RoboDK station: 1817972 amirah husna manual.rdk

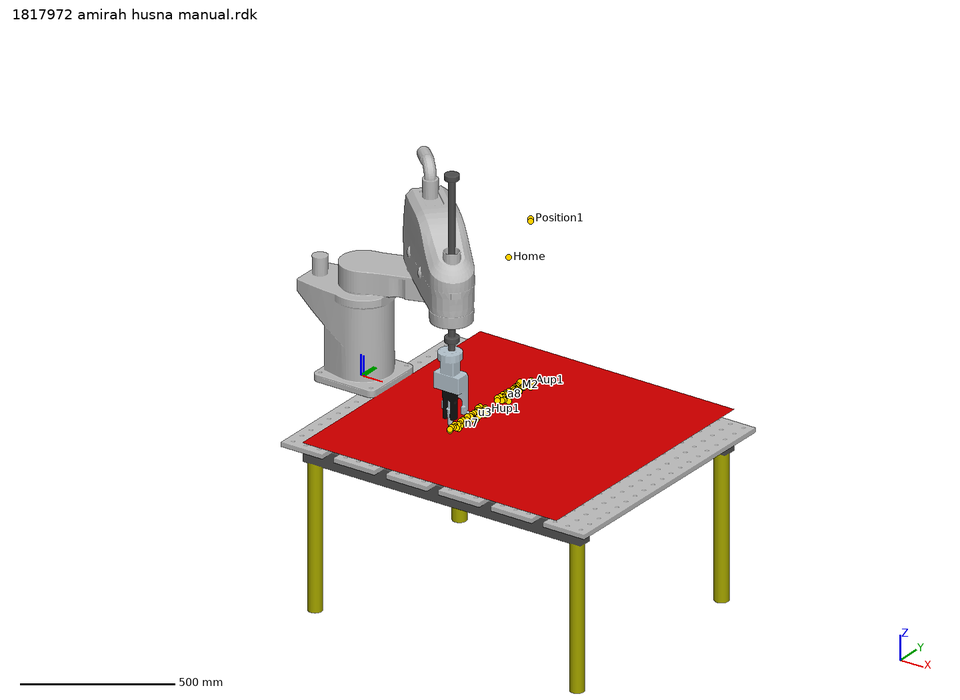
[picture v0: the station drawn from its stored meshes, robots at their saved joint values, targets as dots, program paths as lines]
Station amirah husna manual (saved by RoboDK 5.3.4). Poses are relative to the parent item; angles as X-Y-Z fixed-axis rotations.
  - frame Mitsubishi RH-12SH5535 Base at (0, 0, 0) mm
    - robot Mitsubishi RH-12SH5535: 4 axes, payload 12 kg, reach 600 mm, repeatability 0.03 mm, weight 43 kg
        modified DH rows (alpha deg, a mm, theta deg, d mm): 0, 0, 0, 0; 0, 225, 0, 0; 0, 325, 0, 0 linear; 180, 0, 0, 0
        joint limits [-140, -145, -10, -360] to [140, 145, 340, 360]; home [0, 0, 340, 0]; saved at [18.314, -60.92, 280.095, 42.606]
      - tool Gripper with pencil, TCP at (0, -10, -280) mm, rotated rx 180 ry 0 rz 0 deg, size 100 x 89.2 x 281.5 mm
  - frame Frame 2 at (-10, 0, 0) mm
    - object Object Table at (620, 0, -40) mm, size 1193.8 x 965.2 x 609.6 mm, geometry from Object Table.wrl
    - object Plane at (630, 0, 2) mm, size 1000 x 1000 x 0.5 mm, geometry from plane.sld
    - target Home (Cartesian target) at (557.97, 35.03, 564.41) mm; joints [7.617, -6.699, 291.409, -0.918] of Mitsubishi RH-12SH5535
    - target Aup1 (Cartesian target) at (473.2, 285.09, -0.83) mm, rotated rx 180 ry 0 rz 0 deg; joints [36.19, -6.243, 279.167, -29.946] of Mitsubishi RH-12SH5535
    - target A4 (Cartesian target) at (473.25, 285.09, -5.59) mm, rotated rx 180 ry 0 rz 0 deg; joints [36.081, -6.065, 274.409, -30.016] of Mitsubishi RH-12SH5535
    - target A5 (Cartesian target) at (473.25, 245.06, -5.59) mm, rotated rx 180 ry 0 rz 0 deg; joints [48.093, -32.454, 274.409, -15.638] of Mitsubishi RH-12SH5535
    - target Aup2 (Cartesian target) at (473.14, 245.06, 1.51) mm, rotated rx 180 ry 0 rz 0 deg; joints [48.146, -32.534, 281.511, -15.613] of Mitsubishi RH-12SH5535
    - target Position1 (Cartesian target) at (451.34, 310.3, 564.41) mm; joints [40.788, -10.621, 281.409, -30.167] of Mitsubishi RH-12SH5535
    - target Down1 (Cartesian target) at (451.34, 310.3, 554.41) mm; joints [48.613, -22.805, 281.409, -25.808] of Mitsubishi RH-12SH5535
    - target A1 (Cartesian target) at (493.02, 251.45, -5.59) mm, rotated rx 180 ry 0 rz 0 deg; joints [32.04, -6.116, 274.409, -25.924] of Mitsubishi RH-12SH5535
    - target A2 (Cartesian target) at (451.34, 251.57, -5.59) mm, rotated rx 180 ry 0 rz 0 deg; joints [56.255, -43.006, 274.409, -13.248] of Mitsubishi RH-12SH5535
    - target A3 (Cartesian target) at (456.2, 244.79, -5.59) mm, rotated rx 180 ry 0 rz 0 deg; joints [55.046, -42.54, 274.409, -12.506] of Mitsubishi RH-12SH5535
    - target Aup3 (Cartesian target) at (456.71, 244.79, 6.07) mm, rotated rx 180 ry 0 rz 0 deg; joints [54.857, -42.274, 286.074, -12.583] of Mitsubishi RH-12SH5535
    - target Mup1 (Cartesian target) at (476.08, 240.53, 3.16) mm, rotated rx 180 ry 0 rz 0 deg; joints [47.367, -32.207, 283.156, -15.16] of Mitsubishi RH-12SH5535
    - target M1 (Cartesian target) at (474.44, 240.53, -5.59) mm, rotated rx 180 ry 0 rz 0 deg; joints [48.113, -33.312, 274.409, -14.801] of Mitsubishi RH-12SH5535
    - target M2 (Cartesian target) at (451.34, 237.47, -5.59) mm, rotated rx 180 ry 0 rz 0 deg; joints [57.291, -46.985, 274.409, -10.306] of Mitsubishi RH-12SH5535
    - target M3 (Cartesian target) at (474.44, 230.54, -5.59) mm, rotated rx 180 ry 0 rz 0 deg; joints [49.16, -36.663, 274.409, -12.496] of Mitsubishi RH-12SH5535
    - target M4 (Cartesian target) at (451.34, 230.52, -5.59) mm, rotated rx 180 ry 0 rz 0 deg; joints [57.69, -48.777, 274.409, -8.913] of Mitsubishi RH-12SH5535
    - target M5 (Cartesian target) at (474.44, 219.74, -5.59) mm, rotated rx 180 ry 0 rz 0 deg; joints [50.032, -39.877, 274.409, -10.155] of Mitsubishi RH-12SH5535
    - target M6 (Cartesian target) at (451.34, 219.84, -5.59) mm, rotated rx 180 ry 0 rz 0 deg; joints [58.175, -51.343, 274.409, -6.833] of Mitsubishi RH-12SH5535
    - target M7 (Cartesian target) at (461.93, 215.03, -5.59) mm, rotated rx 180 ry 0 rz 0 deg; joints [54.851, -47.594, 274.409, -7.257] of Mitsubishi RH-12SH5535
    - target I1 (Cartesian target) at (472.85, 204.97, -5.59) mm, rotated rx 180 ry 0 rz 0 deg; joints [51.459, -44.57, 274.41, -6.889] of Mitsubishi RH-12SH5535
    - target I2 (Cartesian target) at (464.34, 211.06, -5.59) mm, rotated rx 180 ry 0 rz 0 deg; joints [54.191, -47.371, 274.41, -6.82] of Mitsubishi RH-12SH5535
    - target I3 (Cartesian target) at (451.34, 211.86, -5.59) mm, rotated rx 180 ry 0 rz 0 deg; joints [58.448, -53.129, 274.409, -5.318] of Mitsubishi RH-12SH5535
    - target I4 (Cartesian target) at (461.93, 203.58, -5.59) mm, rotated rx 180 ry 0 rz 0 deg; joints [55.266, -50.203, 274.409, -5.063] of Mitsubishi RH-12SH5535
    - target R1 (Cartesian target) at (470.19, 197.42, -5.59) mm, rotated rx 180 ry 0 rz 0 deg; joints [52.669, -47.637, 274.409, -5.033] of Mitsubishi RH-12SH5535
    - target R2 (Cartesian target) at (477.11, 195.12, -5.59) mm, rotated rx 180 ry 0 rz 0 deg; joints [50.312, -44.666, 274.409, -5.646] of Mitsubishi RH-12SH5535
    - target R3 (Cartesian target) at (469.73, 199.31, -5.59) mm, rotated rx 180 ry 0 rz 0 deg; joints [52.767, -47.441, 274.409, -5.326] of Mitsubishi RH-12SH5535
    - target R3.5 (Cartesian target) at (469.73, 201.5, -5.59) mm, rotated rx 180 ry 0 rz 0 deg; joints [52.694, -46.948, 274.409, -5.746] of Mitsubishi RH-12SH5535
    - target R3.55 (Cartesian target) at (471.65, 195.27, -5.59) mm, rotated rx 180 ry 0 rz 0 deg; joints [52.233, -47.396, 274.409, -4.836] of Mitsubishi RH-12SH5535
    - target R3.6 (Cartesian target) at (471.65, 190.99, -5.59) mm, rotated rx 180 ry 0 rz 0 deg; joints [52.346, -48.315, 274.409, -4.032] of Mitsubishi RH-12SH5535
    - target R4 (Cartesian target) at (474.41, 185.39, -5.59) mm, rotated rx 180 ry 0 rz 0 deg; joints [51.527, -48.134, 274.409, -3.393] of Mitsubishi RH-12SH5535
    - target R5 (Cartesian target) at (461.56, 188.8, -5.59) mm, rotated rx 180 ry 0 rz 0 deg; joints [55.692, -53.409, 274.409, -2.283] of Mitsubishi RH-12SH5535
    - target R6 (Cartesian target) at (451.34, 186.17, -5.59) mm, rotated rx 180 ry 0 rz 0 deg; joints [58.859, -58.225, 274.409, -0.634] of Mitsubishi RH-12SH5535
    - target R7 (Cartesian target) at (461.93, 176.77, -5.59) mm, rotated rx 180 ry 0 rz 0 deg; joints [55.657, -55.483, 274.409, -0.174] of Mitsubishi RH-12SH5535
    - target a1 (Cartesian target) at (471.07, 162.8, -5.59) mm, rotated rx 180 ry 0 rz 0 deg; joints [52.77, -53.89, 274.409, 1.12] of Mitsubishi RH-12SH5535
    - target a2 (Cartesian target) at (476.85, 158.23, -5.59) mm, rotated rx 180 ry 0 rz 0 deg; joints [50.897, -52.02, 274.409, 1.123] of Mitsubishi RH-12SH5535
    - target a3 (Cartesian target) at (459.52, 173.46, -5.59) mm, rotated rx 180 ry 0 rz 0 deg; joints [56.39, -57.081, 274.409, 0.692] of Mitsubishi RH-12SH5535
    - target a4 (Cartesian target) at (451.34, 169.13, -5.59) mm, rotated rx 180 ry 0 rz 0 deg; joints [58.784, -61.128, 274.409, 2.345] of Mitsubishi RH-12SH5535
    - target a5 (Cartesian target) at (460.8, 160.64, -5.59) mm, rotated rx 180 ry 0 rz 0 deg; joints [55.888, -58.649, 274.409, 2.76] of Mitsubishi RH-12SH5535
    - target a6 (Cartesian target) at (470.78, 157.7, -5.59) mm, rotated rx 180 ry 0 rz 0 deg; joints [52.816, -54.853, 274.409, 2.037] of Mitsubishi RH-12SH5535
    - target a7 (Cartesian target) at (457.33, 158.29, -5.59) mm, rotated rx 180 ry 0 rz 0 deg; joints [56.875, -60.428, 274.409, 3.553] of Mitsubishi RH-12SH5535
    - target a8 (Cartesian target) at (451.34, 154.04, -5.59) mm, rotated rx 180 ry 0 rz 0 deg; joints [58.509, -63.419, 274.409, 4.91] of Mitsubishi RH-12SH5535
    - target a9 (Cartesian target) at (461.93, 142.7, -5.59) mm, rotated rx 180 ry 0 rz 0 deg; joints [55.169, -60.819, 274.409, 5.65] of Mitsubishi RH-12SH5535
    - target h1 (Cartesian target) at (493.02, 127.33, -5.59) mm, rotated rx 180 ry 0 rz 0 deg; joints [45.116, -49.014, 274.409, 3.898] of Mitsubishi RH-12SH5535
    - target h2 (Cartesian target) at (461.93, 139.05, -5.59) mm, rotated rx 180 ry 0 rz 0 deg; joints [55.059, -61.311, 274.409, 6.252] of Mitsubishi RH-12SH5535
    - target h3 (Cartesian target) at (451.34, 136.81, -5.59) mm, rotated rx 180 ry 0 rz 0 deg; joints [57.972, -65.744, 274.409, 7.771] of Mitsubishi RH-12SH5535
    - target h4 (Cartesian target) at (477.38, 125.53, -5.59) mm, rotated rx 180 ry 0 rz 0 deg; joints [50.045, -56.573, 274.409, 6.528] of Mitsubishi RH-12SH5535
    - target h5 (Cartesian target) at (473.98, 118.78, -5.59) mm, rotated rx 180 ry 0 rz 0 deg; joints [50.804, -58.868, 274.409, 8.065] of Mitsubishi RH-12SH5535
    - target h6 (Cartesian target) at (451.34, 123.67, -5.59) mm, rotated rx 180 ry 0 rz 0 deg; joints [57.412, -67.317, 274.409, 9.905] of Mitsubishi RH-12SH5535
    - target h7 (Cartesian target) at (461.93, 108.73, -5.59) mm, rotated rx 180 ry 0 rz 0 deg; joints [53.751, -64.879, 274.409, 11.128] of Mitsubishi RH-12SH5535
    - target Updot1 (Cartesian target) at (483.42, 201.03, -1.25) mm, rotated rx 180 ry 0 rz 0 deg; joints [47.671, -39.768, 278.753, -7.903] of Mitsubishi RH-12SH5535
    - target Dot1 (Cartesian target) at (483.71, 201.03, -5.59) mm, rotated rx 180 ry 0 rz 0 deg; joints [47.559, -39.602, 274.41, -7.956] of Mitsubishi RH-12SH5535
    - target Dot2 (Cartesian target) at (482.8, 201.03, -5.59) mm, rotated rx 180 ry 0 rz 0 deg; joints [47.916, -40.127, 274.41, -7.788] of Mitsubishi RH-12SH5535
    - target Updot2 (Cartesian target) at (482.51, 201.03, -2.21) mm, rotated rx 180 ry 0 rz 0 deg; joints [48.028, -40.293, 277.786, -7.736] of Mitsubishi RH-12SH5535
    - target Hup1 (Cartesian target) at (476.08, 28.37, 0.73) mm, rotated rx 180 ry 0 rz 0 deg; joints [43.638, -64.719, 280.727, 21.082] of Mitsubishi RH-12SH5535
    - target H1 (Cartesian target) at (476.67, 28.37, -5.59) mm, rotated rx 180 ry 0 rz 0 deg; joints [43.484, -64.482, 274.409, 20.999] of Mitsubishi RH-12SH5535
    - target H2 (Cartesian target) at (481.32, 33.14, -5.59) mm, rotated rx 180 ry 0 rz 0 deg; joints [42.714, -62.4, 274.409, 19.686] of Mitsubishi RH-12SH5535
    - target H3 (Cartesian target) at (493.02, 15.59, -5.59) mm, rotated rx 180 ry 0 rz 0 deg; joints [37.726, -57.9, 274.409, 20.174] of Mitsubishi RH-12SH5535
    - target H4 (Cartesian target) at (486.33, 12.57, -5.59) mm, rotated rx 180 ry 0 rz 0 deg; joints [39.258, -60.89, 274.409, 21.632] of Mitsubishi RH-12SH5535
    - target H5 (Cartesian target) at (451.34, 26.46, -5.59) mm, rotated rx 180 ry 0 rz 0 deg; joints [49.642, -74.184, 274.409, 24.542] of Mitsubishi RH-12SH5535
    - target Hup2 (Cartesian target) at (451.16, 26.46, 2.44) mm, rotated rx 180 ry 0 rz 0 deg; joints [49.686, -74.25, 282.435, 24.564] of Mitsubishi RH-12SH5535
    - target Hup3 (Cartesian target) at (452.87, 11.87, 5.16) mm, rotated rx 180 ry 0 rz 0 deg; joints [47.616, -73.981, 285.163, 26.365] of Mitsubishi RH-12SH5535
    - target H6 (Cartesian target) at (451.34, 11.87, -5.59) mm, rotated rx 180 ry 0 rz 0 deg; joints [47.978, -74.531, 274.409, 26.553] of Mitsubishi RH-12SH5535
    - target H7 (Cartesian target) at (454.28, 14.58, -5.59) mm, rotated rx 180 ry 0 rz 0 deg; joints [47.595, -73.417, 274.409, 25.821] of Mitsubishi RH-12SH5535
    - target H8 (Cartesian target) at (490.19, 1.69, -5.59) mm, rotated rx 180 ry 0 rz 0 deg; joints [37.009, -59.39, 274.409, 22.381] of Mitsubishi RH-12SH5535
    - target Hup4 (Cartesian target) at (489.79, 1.69, -0.69) mm, rotated rx 180 ry 0 rz 0 deg; joints [37.119, -59.566, 279.311, 22.447] of Mitsubishi RH-12SH5535
    - target Hup5 (Cartesian target) at (466.33, 33.1, 0.85) mm, rotated rx 180 ry 0 rz 0 deg; joints [46.638, -68.398, 280.846, 21.76] of Mitsubishi RH-12SH5535
    - target H9 (Cartesian target) at (466.14, 33.1, -5.59) mm, rotated rx 180 ry 0 rz 0 deg; joints [46.687, -68.472, 274.409, 21.785] of Mitsubishi RH-12SH5535
    - target H10 (Cartesian target) at (469.45, 20.76, -5.59) mm, rotated rx 180 ry 0 rz 0 deg; joints [44.555, -67.576, 274.409, 23.022] of Mitsubishi RH-12SH5535
    - target H11 (Cartesian target) at (472.39, 2.61, -5.59) mm, rotated rx 180 ry 0 rz 0 deg; joints [41.773, -66.759, 274.409, 24.986] of Mitsubishi RH-12SH5535
    - target Hup6 (Cartesian target) at (471.59, 2.61, 2.6) mm, rotated rx 180 ry 0 rz 0 deg; joints [41.974, -67.074, 282.598, 25.1] of Mitsubishi RH-12SH5535
    - target uup1 (Cartesian target) at (476.74, -11.13, -1.91) mm, rotated rx 180 ry 0 rz 0 deg; joints [39.026, -65.092, 278.086, 26.065] of Mitsubishi RH-12SH5535
    - target u1 (Cartesian target) at (477.08, -11.13, -5.59) mm, rotated rx 180 ry 0 rz 0 deg; joints [38.939, -64.952, 274.409, 26.013] of Mitsubishi RH-12SH5535
    - target u2 (Cartesian target) at (459.41, -2.79, -5.59) mm, rotated rx 180 ry 0 rz 0 deg; joints [44.294, -71.763, 274.409, 27.469] of Mitsubishi RH-12SH5535
    - target u2.5 (Cartesian target) at (454.9, -4.46, -5.59) mm, rotated rx 180 ry 0 rz 0 deg; joints [45.15, -73.428, 274.409, 28.278] of Mitsubishi RH-12SH5535
    - target u3 (Cartesian target) at (451.34, -11.79, -5.59) mm, rotated rx 180 ry 0 rz 0 deg; joints [45.033, -74.724, 274.409, 29.691] of Mitsubishi RH-12SH5535
    - target u4 (Cartesian target) at (480.93, -23.56, -5.59) mm, rotated rx 180 ry 0 rz 0 deg; joints [36.395, -63.3, 274.409, 26.905] of Mitsubishi RH-12SH5535
    - target u5 (Cartesian target) at (451.34, -24.07, -5.59) mm, rotated rx 180 ry 0 rz 0 deg; joints [43.388, -74.644, 274.409, 31.257] of Mitsubishi RH-12SH5535
    - target u6 (Cartesian target) at (461.93, -36.56, -5.59) mm, rotated rx 180 ry 0 rz 0 deg; joints [39.242, -70.551, 274.409, 31.309] of Mitsubishi RH-12SH5535
    - target s1 (Cartesian target) at (480.93, -50.57, -5.59) mm, rotated rx 180 ry 0 rz 0 deg; joints [32.72, -62.657, 274.409, 29.937] of Mitsubishi RH-12SH5535
    - target s2 (Cartesian target) at (485.98, -46.68, -5.59) mm, rotated rx 180 ry 0 rz 0 deg; joints [31.998, -60.666, 274.409, 28.667] of Mitsubishi RH-12SH5535
    - target s3 (Cartesian target) at (474.44, -57.02, -5.59) mm, rotated rx 180 ry 0 rz 0 deg; joints [33.364, -65.062, 274.409, 31.697] of Mitsubishi RH-12SH5535
    - target s4 (Cartesian target) at (464.69, -51.2, -5.59) mm, rotated rx 180 ry 0 rz 0 deg; joints [36.504, -69.093, 274.409, 32.588] of Mitsubishi RH-12SH5535
    - target s4.5 (Cartesian target) at (454.51, -44.67, -5.59) mm, rotated rx 180 ry 0 rz 0 deg; joints [39.76, -73.091, 274.409, 33.331] of Mitsubishi RH-12SH5535
    - target s5 (Cartesian target) at (459.29, -36.56, -5.59) mm, rotated rx 180 ry 0 rz 0 deg; joints [39.848, -71.537, 274.409, 31.689] of Mitsubishi RH-12SH5535
    - target s6 (Cartesian target) at (451.34, -44.19, -5.59) mm, rotated rx 180 ry 0 rz 0 deg; joints [40.531, -74.25, 274.409, 33.719] of Mitsubishi RH-12SH5535
    - target s7 (Cartesian target) at (461.93, -65.82, -5.59) mm, rotated rx 180 ry 0 rz 0 deg; joints [34.927, -69.546, 274.409, 34.619] of Mitsubishi RH-12SH5535
    - target n1 (Cartesian target) at (474.05, -70.79, -5.59) mm, rotated rx 180 ry 0 rz 0 deg; joints [31.378, -64.575, 274.409, 33.197] of Mitsubishi RH-12SH5535
    - target n2 (Cartesian target) at (461.93, -65.82, -5.59) mm, rotated rx 180 ry 0 rz 0 deg; joints [34.927, -69.546, 274.409, 34.619] of Mitsubishi RH-12SH5535
    - target n3 (Cartesian target) at (451.34, -69.75, -5.59) mm, rotated rx 180 ry 0 rz 0 deg; joints [36.624, -73.27, 274.409, 36.646] of Mitsubishi RH-12SH5535
    - target n4 (Cartesian target) at (481.43, -87.32, -5.59) mm, rotated rx 180 ry 0 rz 0 deg; joints [27.001, -60.521, 274.409, 33.52] of Mitsubishi RH-12SH5535
    - target n5 (Cartesian target) at (477.62, -90.15, -5.59) mm, rotated rx 180 ry 0 rz 0 deg; joints [27.459, -61.919, 274.409, 34.46] of Mitsubishi RH-12SH5535
    - target n6 (Cartesian target) at (451.34, -83.97, -5.59) mm, rotated rx 180 ry 0 rz 0 deg; joints [34.323, -72.491, 274.409, 38.167] of Mitsubishi RH-12SH5535
    - target n7 (Cartesian target) at (461.93, -101.4, -5.59) mm, rotated rx 180 ry 0 rz 0 deg; joints [29.143, -67.34, 274.409, 38.197] of Mitsubishi RH-12SH5535
    - target aa1 (Cartesian target) at (471.07, -112.44, -5.59) mm, rotated rx 180 ry 0 rz 0 deg; joints [25.214, -62.811, 274.409, 37.597] of Mitsubishi RH-12SH5535
    - target aa2 (Cartesian target) at (476.85, -128.9, -5.59) mm, rotated rx 180 ry 0 rz 0 deg; joints [20.94, -58.766, 274.409, 37.826] of Mitsubishi RH-12SH5535
    - target aa3 (Cartesian target) at (459.52, -107.96, -5.59) mm, rotated rx 180 ry 0 rz 0 deg; joints [28.531, -67.733, 274.409, 39.203] of Mitsubishi RH-12SH5535
    - target aa4 (Cartesian target) at (451.34, -115.42, -5.59) mm, rotated rx 180 ry 0 rz 0 deg; joints [28.92, -70.157, 274.409, 41.237] of Mitsubishi RH-12SH5535
    - target aa5 (Cartesian target) at (460.8, -126.49, -5.59) mm, rotated rx 180 ry 0 rz 0 deg; joints [24.96, -65.545, 274.409, 40.585] of Mitsubishi RH-12SH5535
    - target aa6 (Cartesian target) at (470.78, -131.24, -5.59) mm, rotated rx 180 ry 0 rz 0 deg; joints [21.911, -61.062, 274.409, 39.151] of Mitsubishi RH-12SH5535
    - target aa7 (Cartesian target) at (457.33, -133.6, -5.59) mm, rotated rx 180 ry 0 rz 0 deg; joints [24.383, -66.151, 274.409, 41.768] of Mitsubishi RH-12SH5535
    - target aa8 (Cartesian target) at (451.34, -135.54, -5.59) mm, rotated rx 180 ry 0 rz 0 deg; joints [25.245, -68.209, 274.409, 42.964] of Mitsubishi RH-12SH5535
    - target aa9 (Cartesian target) at (461.93, -159.31, -5.59) mm, rotated rx 180 ry 0 rz 0 deg; joints [18.503, -61.277, 274.409, 42.774] of Mitsubishi RH-12SH5535
    - target aaup1 (Cartesian target) at (462.81, -159.31, 0.09) mm, rotated rx 180 ry 0 rz 0 deg; joints [18.314, -60.92, 280.095, 42.606] of Mitsubishi RH-12SH5535
  - Python program Code (listed below)
  - Python program WeldOn (listed below)
  - Python program WeldOff (listed below)

--- Python program Code ---
# Type help("robolink") or help("robodk") for more information
# Press F5 to run the script
# Documentation: https://robodk.com/doc/en/RoboDK-API.html
# Reference:     https://robodk.com/doc/en/PythonAPI/index.html
# Note: It is not required to keep a copy of this file, your python script is saved with the station
from robolink import *    # RoboDK API
from robodk import *      # Robot toolbox
RDK = Robolink()
RDK.RunProgram("WeldOff(-1)")

# Program example:
robot = RDK.Item('',ITEM_TYPE_ROBOT)
target = RDK.Item('Home')
target_pose = target.Pose()
xyz_ref = target_pose.Pos()

p1 = RDK.Item('Position1')
Ad1 = RDK.Item('Down1')
A1 = RDK.Item('A1')
A2 = RDK.Item('A2')
A3 = RDK.Item('A3')
A4 = RDK.Item('A4')
A5 = RDK.Item('A5')
Aup1 = RDK.Item('Aup1')
Aup2 = RDK.Item('Aup2')
Aup3 = RDK.Item('Aup3')

Mup1 = RDK.Item('Mup1')
M1 = RDK.Item('M1')
M2 = RDK.Item('M2')
M3 = RDK.Item('M3')
M4 = RDK.Item('M4')
M5 = RDK.Item('M5')
M6 = RDK.Item('M6')
M7 = RDK.Item('M7')

I1 = RDK.Item('I1')
I2 = RDK.Item('I2')
I3 = RDK.Item('I3')
I4 = RDK.Item('I4')

R1 = RDK.Item('R1')
R2 = RDK.Item('R2')
R3 = RDK.Item('R3')
R35 = RDK.Item('R3.5')
R355 = RDK.Item('R3.55')
R36 = RDK.Item('R3.6')
R4 = RDK.Item('R4')
R5 = RDK.Item('R5')
R6 = RDK.Item('R6')
R7 = RDK.Item('R7')

a1 = RDK.Item('a1')
a2 = RDK.Item('a2')
a3 = RDK.Item('a3')
a4 = RDK.Item('a4')
a5 = RDK.Item('a5')
a6 = RDK.Item('a6')
a7 = RDK.Item('a7')
a8 = RDK.Item('a8')
a9 = RDK.Item('a9')

h1 = RDK.Item('h1')
h2 = RDK.Item('h2')
h3 = RDK.Item('h3')
h4 = RDK.Item('h4')
h5 = RDK.Item('h5')
h6 = RDK.Item('h6')
h7 = RDK.Item('h7')

H1 = RDK.Item('H1')
H2 = RDK.Item('H2')
H3 = RDK.Item('H3')
H4 = RDK.Item('H4')
H5 = RDK.Item('H5')
H6 = RDK.Item('H6')
H7 = RDK.Item('H7')
H8 = RDK.Item('H8')
H9 = RDK.Item('H10')
H10 = RDK.Item('H10')
H11 = RDK.Item('H11')
Hup1 = RDK.Item('Hup1')
Hup2 = RDK.Item('Hup2')
Hup3 = RDK.Item('Hup3')
Hup4 = RDK.Item('Hup4')
Hup5 = RDK.Item('Hup5')
Hup6 = RDK.Item('Hup6')

uup1 = RDK.Item('uup1')
u1 = RDK.Item('u1')
u2 = RDK.Item('u2')
u3 = RDK.Item('u3')
u4 = RDK.Item('u4')
u5 = RDK.Item('u5')
u6 = RDK.Item('u6')

s1 = RDK.Item('s1')
s2 = RDK.Item('s2')
s3 = RDK.Item('s3')
s4 = RDK.Item('s4')
s45 = RDK.Item('s4.5')
s5 = RDK.Item('s5')
s6 = RDK.Item('s6')
s7 = RDK.Item('s7')

n1 = RDK.Item('n1')
n2 = RDK.Item('n2')
n3 = RDK.Item('n3')
n4 = RDK.Item('n4')
n5 = RDK.Item('n5')
n6 = RDK.Item('n6')
n7 = RDK.Item('n7')

aa1 = RDK.Item('aa1')
aa2 = RDK.Item('aa2')
aa3 = RDK.Item('aa3')
aa4 = RDK.Item('aa4')
aa5 = RDK.Item('aa5')
aa6 = RDK.Item('aa6')
aa7 = RDK.Item('aa7')
aa8 = RDK.Item('aa8')
aa9 = RDK.Item('aa9')
aaup1 = RDK.Item('aaup1')

#dot
updot1 = RDK.Item('Updot1')
updot2 = RDK.Item('Updot2')
dot1 = RDK.Item('Dot1')
dot2 = RDK.Item('Dot2')

fram = RDK.Item('Frame 2')
robot.setFrame(fram) #set active frame

#write name

RDK.RunProgram("WeldOff()")
pause(1)

robot.MoveJ(target)
robot.MoveJ(Aup1)
RDK.RunProgram("WeldOn(1)")
pause(1)
robot.MoveJ(A4)
robot.MoveJ(A5)
robot.MoveJ(Aup2)
RDK.RunProgram("WeldOff()")
pause(1)
robot.MoveJ(p1)
robot.MoveJ(Ad1)
RDK.RunProgram("WeldOn(1)")
pause(1)
robot.MoveJ(A1)
robot.MoveJ(A2)
robot.MoveJ(A3)
RDK.RunProgram("WeldOff()")
pause(1)
robot.MoveJ(Aup3)

robot.MoveJ(Mup1)
RDK.RunProgram("WeldOn(1)")
pause(1)
robot.MoveJ(M1)
robot.MoveJ(M2)
robot.MoveJ(M3)
robot.MoveJ(M4)
robot.MoveJ(M5)
robot.MoveJ(M6)
robot.MoveJ(M7)

robot.MoveJ(I1)
robot.MoveJ(I2)
robot.MoveJ(I3)
robot.MoveJ(I4)

robot.MoveJ(R1)
robot.MoveJ(R2)
robot.MoveJ(R3)
robot.MoveJ(R35)
pause(1)
robot.MoveJ(R355)
robot.MoveJ(R36)
robot.MoveJ(R4)
robot.MoveJ(R5)
robot.MoveJ(R6)
robot.MoveJ(R7)

robot.MoveJ(a1)
robot.MoveJ(a2)
robot.MoveJ(a3)
robot.MoveJ(a4)
robot.MoveJ(a5)
robot.MoveJ(a6)
robot.MoveJ(a7)
robot.MoveJ(a8)
robot.MoveJ(a9)

robot.MoveJ(h1)
robot.MoveJ(h2)
robot.MoveJ(h3)
robot.MoveJ(h4)
robot.MoveJ(h5)
robot.MoveJ(h6)
robot.MoveJ(h7)

RDK.RunProgram("WeldOff()")
pause(1)
robot.MoveJ(updot1)
RDK.RunProgram("WeldOn(1)")
pause(1)
robot.MoveJ(dot1)
robot.MoveJ(dot2)
RDK.RunProgram("WeldOff()")
pause(1)
robot.MoveJ(updot2)

robot.MoveJ(Hup1)
robot.MoveJ(H1)
RDK.RunProgram("WeldOn(1)")
pause(1)
robot.MoveJ(H2)
robot.MoveJ(H3)
robot.MoveJ(H4)
robot.MoveJ(H5)
RDK.RunProgram("WeldOff()")
pause(1)
robot.MoveJ(Hup2)

robot.MoveJ(Hup3)
RDK.RunProgram("WeldOn(1)")
pause(1)
robot.MoveJ(H6)
robot.MoveJ(H7)
robot.MoveJ(H8)
RDK.RunProgram("WeldOff()")
pause(1)
robot.MoveJ(Hup4)

robot.MoveJ(Hup5)
RDK.RunProgram("WeldOn(1)")
pause(1)
robot.MoveJ(H9)
robot.MoveJ(H10)
robot.MoveJ(H11)
RDK.RunProgram("WeldOff()")
pause(1)
robot.MoveJ(Hup6)

robot.MoveJ(uup1)
RDK.RunProgram("WeldOn(1)")
pause(1)
robot.MoveJ(u1)
robot.MoveJ(u2)
robot.MoveJ(u3)
robot.MoveJ(u4)
robot.MoveJ(u5)
robot.MoveJ(u6)

robot.MoveJ(s1)
robot.MoveJ(s2)
robot.MoveJ(s3)
robot.MoveJ(s4)
robot.MoveJ(s45)
robot.MoveJ(s5)
robot.MoveJ(s6)
robot.MoveJ(s7)

robot.MoveJ(n1)
robot.MoveJ(n2)
robot.MoveJ(n3)
robot.MoveJ(n4)
robot.MoveJ(n5)
robot.MoveJ(n6)
robot.MoveJ(n7)

robot.MoveJ(aa1)
robot.MoveJ(aa2)
robot.MoveJ(aa3)
robot.MoveJ(aa4)
robot.MoveJ(aa5)
robot.MoveJ(aa6)
robot.MoveJ(aa7)
robot.MoveJ(aa8)
robot.MoveJ(aa9)
robot.MoveJ(aaup1)

pause(1)

--- Python program WeldOn ---
# This macro allows simulating the material deposition of a weld gun
# By default, this macro will activate the trace once it is called.
# Run the macro ArcEnd to stop the trace.
#
# The macros ArcStart, ArcEnd and WeldOn, SpindleOn, all behave in a similar way, the only difference is the default behavior
# This behavior simmulates Fanuc Arc Welding and triggers appropriate output when using the customized post processor.
# Select ESC to clear the trace manually.
#
# It is possible to call WeldOn(ON) to simulate turning the material deposition ON or WeldOn(OFF) to stop simulating the gun
# Calling WeldOn(RESET) clears all displayed data.
# The macro will output spray gun statistics
#
# Optional:
#     This macro can manage multiple guns and multiple colors.
#     As an example, you can call this macro the following way:
#
# WeldOn(State, ToolName, Color)
#     State: [ON/OFF/RESET]
#     TorchName: The name of the tool. For example: Tool 1
#     Color: A named color or a hex color in the format: '#AARRGGBB'
#             Important: for full color definition you should provide Alpha channel first
#
# Examples:
#     WeldOn(ON)                 # Turn on the trace using the default color
#     WeldOn(OFF)                # Turn off the tool trace
#     WeldOn(ON, Tool 1, yellow) # Turn on the trace for tool 1 in yellow
#     WeldOn(ON, Tool 2, blue) # Turn on the trace for tool 2 in blue
#     WeldOn(OFF, Torch1)        # Turn off trace for Torch 1
#     WeldOn(ON, Torch1, #889900FF) # Turn on the trace for torch 2 in a violet color
#     WeldOn(ON, ,red)         # Turn on the trace for a generic torch in red color
#
# --------------------------------------------------------------
# This script shows how to create "spray" object in RoboDK that allows simulating particle deposition by using:
# RDK.Spray_Add(tool, object, options_command, volume, geometry)
#    tool: tool item (TCP) to use
#    object: object to project the particles
#    options_command (optional): string to specify options.
#    volume (optional): Matrix of parameters defining the volume of the spray gun
#    geometry (optional): Matrix of vertices defining the triangles.
#
# More information here:
# https://robodk.com/doc/en/PythonAPI/robolink.html#robolink.Robolink.Spray_Add
# https://robodk.com/doc/en/RoboDK-API.html
#
# The scripts ArcStart, ArcEnd and WeldOn and SpindleOn behave in a similar way, the only difference is the default behavior
# This behavior simmulates Fanuc Arc Welding and triggers appropriate output when using the customized post processor.
# Select ESC to clear the trace manually.
#
# Example scripts that use Spray_Add:
#     SpindleOn / SpindleOff    -> Turn trace On/Off
#     ArcOn / ArcOff            -> Turn trace On/Off
#     SprayOn / SprayOff        -> Simulate a spray given a workspace volume (for painting)
#     WeldOn / WeldOff          -> Support for multiple weld guns
#
#----------------------------------------------------------

# Constant variables for the first parameter:
ACTION_RESET    = -1    # Same as: RESET (clear all traces)
ACTION_OFF      =  0    # Same as: OFF (turn on)
ACTION_ON       =  1    # Same as: ON (turn off)

# Define the default Action (ACTION_OFF to deactivate, ACTION_ON to activate, ACTION_RESET to clear any spray gun/trace)
# Setting it to None will display a message
Action = ACTION_ON

# Define the default color as a named color or as #AARRGGBB (Alpha, Red, Green Blue)
# COLOR = 'blue'
COLOR = '#CC3344FF' # AARRGGBB

# Use a specific tool as a spray gun
Tool_Name = None    # Use the active tool
#Tool_Name = 'Torch1'

# Use a specific object to project particles:
Object_Name = None  # Use the first object in the active reference frame
#Object_Name = 'Part'

# --------------------------------------------------
# Program start:
from robolink import *    # API to communicate with RoboDK
from robodk import *      # basic matrix operations
RDK = Robolink()

# quit if we are not in simulation mode
if RDK.RunMode() != RUNMODE_SIMULATE:
    quit()

# Check command input (parameters passed in the call). This is the same as if we were doing a command line call passing parameters.
import sys
if len(sys.argv) > 1:
    Action_str = sys.argv[1].strip().upper()
    if 'ON' in Action_str:
        Action = ACTION_ON
    elif 'OFF' in Action_str:
        Action = ACTION_OFF
    elif 'RESET' in Action_str:
        Action = ACTION_RESET
    else:
        Action = int(Action_str)

    if len(sys.argv) > 2:
        Tool_Name = sys.argv[2].strip()
        if Tool_Name == '':
            Tool_Name = None

        if len(sys.argv) > 3:
            COLOR = sys.argv[3].lower().strip()

# Display summary
print("Applying action: " + str(Action))
print("Using tool: " + str(Tool_Name))
print("Using color: " + COLOR)

# Get any previously added spray gun simulations and display statistics (spray on the part vs spray falling out of the part)
info, data = RDK.Spray_GetStats()
n_sprays = data.size(1)
spray_id = -1
if n_sprays > 0 and Tool_Name is not None:
    spray_id = RDK.getParam(Tool_Name)
    if spray_id is None or Action == ACTION_ON or type(spray_id) == str or spray_id >= n_sprays:
        spray_id = -1

    print("Spray gun statistics:")
    print(info)
    print(data.tr())
    # # Diplay statistics
    # RDK.ShowMessage("Material used: %.1f%%<br>Material waisted: %.1f%%<br>Total particles: %.1f" % (data[1,0],data[2,0],data[3,0]), True)
    # # Clear previous spray
    # RDK.Spray_Clear()


# If the default Action is None, display a message to activate/deactivate the spray gun
if Action is None:
    print('Note: This macro can be called as ArcStart(1) or ArcStart(0) or ArcStart(-1)')
    entry = mbox('Turn gun ON or OFF', ('On', '1'), ('Off', '0'))
    if not entry:
        quit()
    Action = int(entry)

# Apply the desired action
if Action == ACTION_OFF:
    # Turn the gun off
    RDK.Spray_SetState(SPRAY_OFF, spray_id)

elif Action == ACTION_OFF:
    # Clear all spray simulations (same as pressing ESC key)
    RDK.Spray_Clear(spray_id)

elif Action == ACTION_ON:
    # Create a new spray gun object in RoboDK
    # by using RDK.Spray_Add(tool, object, options_command, volume, geometry)
    # tool: tool item (TCP) to use
    # object: object to project the particles
    # options_command (optional): string to specify options. Example:
    #     STEP=AxB: Defines the grid to be projected 1x1 means only one line of particle projection (for example, for welding)
    #     PARTICLE: Defines the shape and size of particle (sphere or particle), unless a specific geometry is provided:
    #       a- SPHERE(radius, facets)
    #       b- SPHERE(radius, facets, scalex, scaley, scalez)
    #       b- CUBE(sizex, sizey, sizez)
    #     RAND=factor: Defines a random factor factor 0 means that the particles are not deposited randomly
    #     ELLYPSE: defines the volume as an ellypse (default)
    #     RECTANGLE: defines the volume as a rectangle
    #     PROJECT: project the particles to the surface (default) (for welding, painting or scanning)
    #     NO_PROJECT: does not project the particles to the surface (for example, for 3D printing)
    #
    # volume (optional): Matrix of parameters defining the volume of the spray gun
    # geometry (optional): Matrix of vertices defining the triangles.

    if spray_id < 0:
        tool = 0    # auto detect active tool
        obj = 0     # auto detect object in active reference frame
        if Tool_Name is not None:
            tool = RDK.Item(Tool_Name, ITEM_TYPE_TOOL)

        if Object_Name is not None:
            obj = RDK.Item(Object_Name, ITEM_TYPE_OBJECT)
        # We can specify a given tool object and/or object
        #robot = RDK.Item("ABB IRB 2600-12/1.85", ITEM_TYPE_ROBOT)
        #tools = robot.Childs()
        #if len(tools) > 0:
        #    tool = tools[0]
        #obj = RDK.Item('object', ITEM_TYPE_OBJECT)

        # Create volume parameters
        options_command = "NO_PROJECT PARTICLE=SPHERE(2,8,1,1,1) STEP=1x0 RAND=0 COLOR=" + COLOR

        spray_id = RDK.Spray_Add(tool, obj, options_command)

    # Remember the ID of the spray gun for later
    if Tool_Name is not None:
        RDK.setParam(Tool_Name, spray_id)

    # Apply the state to activate the trace
    RDK.Spray_SetState(SPRAY_ON, spray_id)

--- Python program WeldOff ---
# This macro allows simulating the material deposition of a weld gun
# By default, this macro will activate the trace once it is called.
# Run the macro ArcEnd to stop the trace.
#
# The macros WeldOn, ArcEnd and Arc, all behave the same way, the only difference is the default behavior
# This behavior simmulates Fanuc Arc Welding and triggers appropriate output when using the customized post processor.
# Select ESC to clear the trace manually.
#
# It is possible to call WeldOn(ON) to simulate turning the material deposition ON or WeldOn(OFF) to stop simulating the gun
# Calling WeldOn(RESET) clears all displayed data.
# The macro will output spray gun statistics
#
# Optional:
# This macro can manage multiple guns and multiple colors.
# As an example, you can call this macro the following way:
#
# AcrStart(State, ToolName, Color)
#     State: [ON/OFF/RESET]
#     TorchName: The name of the tool. For example: Tool 1
#     Color: A named color or a hex color in the format: '#AARRGGBB'
#             Important: for full color definition you should provide Alpha channel first
#
# Examples:
#     WeldOn(ON)                 # Turn on the trace using the default color
#     WeldOn(OFF)                # Turn off the tool trace
#     WeldOn(ON, Tool 1, yellow) # Turn on the trace for tool 1 in yellow
#     WeldOn(ON, Tool 2, blue) # Turn on the trace for tool 2 in blue
#     WeldOn(OFF, Torch1)        # Turn off trace for Torch 1
#     WeldOn(ON, Torch1, #889900FF) # Turn on the trace for torch 2 in a violet color
#     WeldOn(ON, ,red)         # Turn on the trace for a generic torch in red color
#
# --------------------------------------------------------------
# This script shows how to create "spray" object in RoboDK that allows simulating particle deposition by using:
# RDK.Spray_Add(tool, object, options_command, volume, geometry)
#    tool: tool item (TCP) to use
#    object: object to project the particles
#    options_command (optional): string to specify options.
#    volume (optional): Matrix of parameters defining the volume of the spray gun
#    geometry (optional): Matrix of vertices defining the triangles.
#
# More information here:
# https://robodk.com/doc/en/PythonAPI/robolink.html#robolink.Robolink.Spray_Add
# https://robodk.com/doc/en/RoboDK-API.html
#
# The scripts ArcStart, ArcEnd and WeldOn and SpindleOn behave in a similar way, the only difference is the default behavior
# This behavior simmulates Fanuc Arc Welding and triggers appropriate output when using the customized post processor.
# Select ESC to clear the trace manually.
#
# Example scripts that use Spray_Add:
#     SpindleOn / SpindleOff    -> Turn trace On/Off
#     ArcOn / ArcOff            -> Turn trace On/Off
#     SprayOn / SprayOff        -> Simulate a spray given a workspace volume (for painting)
#     WeldOn / WeldOff          -> Support for multiple weld guns
#
#----------------------------------------------------------

# Constant variables for the first parameter:
ACTION_RESET    = -1    # Same as: RESET (clear all traces)
ACTION_OFF      =  0    # Same as: OFF (turn on)
ACTION_ON       =  1    # Same as: ON (turn off)

# Define the default Action (ACTION_OFF to deactivate, ACTION_ON to activate, ACTION_RESET to clear any spray gun/trace)
# Setting it to None will display a message
Action = ACTION_OFF

# Define the default color as a named color or as #AARRGGBB (Alpha, Red, Green Blue)
# COLOR = 'blue'
COLOR = '#CC3344FF' # AARRGGBB

# Use a specific tool as a spray gun
Tool_Name = None    # Use the active tool
#Tool_Name = 'Torch1'

# Use a specific object to project particles:
Object_Name = None  # Use the first object in the active reference frame
#Object_Name = 'Part'

# --------------------------------------------------
# Program start:
from robolink import *    # API to communicate with RoboDK
from robodk import *      # basic matrix operations
RDK = Robolink()

# quit if we are not in simulation mode
if RDK.RunMode() != RUNMODE_SIMULATE:
    quit()

# Check command input (parameters passed in the call). This is the same as if we were doing a command line call passing parameters.
import sys
if len(sys.argv) > 1:
    Action_str = sys.argv[1].strip().upper()
    if 'ON' in Action_str:
        Action = ACTION_ON
    elif 'OFF' in Action_str:
        Action = ACTION_OFF
    elif 'RESET' in Action_str:
        Action = ACTION_RESET
    else:
        Action = int(Action_str)

    if len(sys.argv) > 2:
        Tool_Name = sys.argv[2].strip()
        if Tool_Name == '':
            Tool_Name = None

        if len(sys.argv) > 3:
            COLOR = sys.argv[3].lower().strip()

# Display summary
print("Applying action: " + str(Action))
print("Using tool: " + str(Tool_Name))
print("Using color: " + COLOR)

# Get any previously added spray gun simulations and display statistics (spray on the part vs spray falling out of the part)
info, data = RDK.Spray_GetStats()
n_sprays = data.size(1)
spray_id = -1
if n_sprays > 0 and Tool_Name is not None:
    spray_id = RDK.getParam(Tool_Name)
    if spray_id is None or Action == ACTION_ON or type(spray_id) == str or spray_id >= n_sprays:
        spray_id = -1

    print("Spray gun statistics:")
    print(info)
    print(data.tr())
    # # Diplay statistics
    # RDK.ShowMessage("Material used: %.1f%%<br>Material waisted: %.1f%%<br>Total particles: %.1f" % (data[1,0],data[2,0],data[3,0]), True)
    # # Clear previous spray
    # RDK.Spray_Clear()


# If the default Action is None, display a message to activate/deactivate the spray gun
if Action is None:
    print('Note: This macro can be called as ArcStart(1) or ArcStart(0) or ArcStart(-1)')
    entry = mbox('Turn gun ON or OFF', ('On', '1'), ('Off', '0'))
    if not entry:
        quit()
    Action = int(entry)

# Apply the desired action
if Action == ACTION_OFF:
    # Turn the gun off
    RDK.Spray_SetState(SPRAY_OFF, spray_id)

elif Action == ACTION_OFF:
    # Clear all spray simulations (same as pressing ESC key)
    RDK.Spray_Clear(spray_id)

elif Action == ACTION_ON:
    # Create a new spray gun object in RoboDK
    # by using RDK.Spray_Add(tool, object, options_command, volume, geometry)
    # tool: tool item (TCP) to use
    # object: object to project the particles
    # options_command (optional): string to specify options. Example:
    #     STEP=AxB: Defines the grid to be projected 1x1 means only one line of particle projection (for example, for welding)
    #     PARTICLE: Defines the shape and size of particle (sphere or particle), unless a specific geometry is provided:
    #       a- SPHERE(radius, facets)
    #       b- SPHERE(radius, facets, scalex, scaley, scalez)
    #       b- CUBE(sizex, sizey, sizez)
    #     RAND=factor: Defines a random factor factor 0 means that the particles are not deposited randomly
    #     ELLYPSE: defines the volume as an ellypse (default)
    #     RECTANGLE: defines the volume as a rectangle
    #     PROJECT: project the particles to the surface (default) (for welding, painting or scanning)
    #     NO_PROJECT: does not project the particles to the surface (for example, for 3D printing)
    #
    # volume (optional): Matrix of parameters defining the volume of the spray gun
    # geometry (optional): Matrix of vertices defining the triangles.

    if spray_id < 0:
        tool = 0    # auto detect active tool
        obj = 0     # auto detect object in active reference frame
        if Tool_Name is not None:
            tool = RDK.Item(Tool_Name, ITEM_TYPE_TOOL)

        if Object_Name is not None:
            obj = RDK.Item(Object_Name, ITEM_TYPE_OBJECT)
        # We can specify a given tool object and/or object
        #robot = RDK.Item("ABB IRB 2600-12/1.85", ITEM_TYPE_ROBOT)
        #tools = robot.Childs()
        #if len(tools) > 0:
        #    tool = tools[0]
        #obj = RDK.Item('object', ITEM_TYPE_OBJECT)

        # Create volume parameters
        options_command = "NO_PROJECT PARTICLE=SPHERE(2,8,1,1,1) STEP=1x0 RAND=0 COLOR=" + COLOR

        spray_id = RDK.Spray_Add(tool, obj, options_command)

    # Remember the ID of the spray gun for later
    if Tool_Name is not None:
        RDK.setParam(Tool_Name, spray_id)

    # Apply the state to activate the trace
    RDK.Spray_SetState(SPRAY_ON, spray_id)
